Staubli VAL3: normal.dtx

frame fUserFrame = {fatherId=world[0]}
jointRx jtPark = {j1=-90, j2=-20, j3=140, j5=-60, j6=178}
public jointRx ptRoutingPath = {j1=10.656, j2=46.412, j3=64.252, j4=10.088, j5=67.637, j6=-59.47}
mdesc mNomSpeed = {blend=off}
public mdesc mdJointBlend = {accel=250, decel=150, leave=1, reach=1}
public mdesc mdLineBlend = {accel=80, vel=60, decel=50, tmax=100, rmax=9999, leave=2, reach=2}
public tool tTool = {x=487, y=64, z=-100.5, rx=5, rz=-92.998, fatherId=flange[0], ioLink=valve1}
